// TIA Portal V19 export
FUNCTION_BLOCK "Prod_HMI_Mng"   // FB194, LAD
TITLE = GESTIONE OPERAZIONI ESEGUITE DA HMI
// stored: MemoryReserve 100, SetENOAutomatically false
   VAR_INPUT
      CTRL_LinePreraration : Bool;
      MODE { ExternalAccessible := 'False'; ExternalVisible := 'False'; ExternalWritable := 'False'} : "Prod_Mode";
      PART_PROD { ExternalWritable := 'False'} : "Prod_Part_Area";
      BEAM_PROD { ExternalWritable := 'False'} : "Prod_Beam_Area";
   END_VAR
   VAR_IN_OUT
      SET_UP : "Prod_SetUp_Data";
   END_VAR
   VAR
      i : Int;
      indx_Detail : Int;
      Sts : Struct
         Enable_Pop_ACT_to_TODO : Bool;
         Sel_TODO_CanBeExecuted : Bool;
      END_STRUCT;
      Ctrl : Struct
         Pop_ACT_to_TODO : Bool;
         "Pop_O_ACT_&_Push_O_ENDING" : Bool;
         "Pop_O_TODO_&_Push_O_ACT" : Bool;
         Push_HMI_Order_Push_O_TODO : Bool;
         Move_O_TODO_UP : Bool;
         Move_O_TODO_DW : Bool;
         "Pop_O_TODO_&_Push_O_ENDING" : Bool;
      END_STRUCT;
      TON_HMI_Pop_ACT_To_TODO : TON_TIME;
      TON_HMI_Clear_Index_TODO { S7_SetPoint := 'True'} : TON_TIME;
      TON_HMI_Pop_ACT_To_ENDING { S7_SetPoint := 'True'} : TON_TIME;
      TON_HMI_Pop_TODO_To_ACT { S7_SetPoint := 'True'} : TON_TIME;
      TON_HMI_Pop_TODO_To_ENDING { S7_SetPoint := 'True'} : TON_TIME;
      O_TODO_Push_ManualOrder_HMI { S7_SetPoint := 'True'} : "Prod_O_TODO_Push_ManualOrder";
      O_TODO_Swap_Positions_HMI { S7_SetPoint := 'True'} : "Prod_O_TODO_Swap_Positions";
      SetUp_Man_Mng { S7_SetPoint := 'True'} : "Prod_SetUp_Man";
      AUX : Struct
         Button_Pop_ACT_To_ENDING { ExternalAccessible := 'False'; ExternalVisible := 'False'; ExternalWritable := 'False'} : Bool;
         Button_Pop_ACT_To_TODO { ExternalAccessible := 'False'; ExternalVisible := 'False'; ExternalWritable := 'False'} : Bool;
         Button_Pop_TODO_To_ACT { ExternalAccessible := 'False'; ExternalVisible := 'False'; ExternalWritable := 'False'} : Bool;
         Button_Push_ManualOrder_To_TODO { ExternalAccessible := 'False'; ExternalVisible := 'False'; ExternalWritable := 'False'} : Bool;
         Button_ChangeOrder_TODO_UP { ExternalAccessible := 'False'; ExternalVisible := 'False'; ExternalWritable := 'False'} : Bool;
         Button_ChangeOrder_TODO_DW { ExternalAccessible := 'False'; ExternalVisible := 'False'; ExternalWritable := 'False'} : Bool;
         Button_Pop_TODO_To_ENDING { ExternalAccessible := 'False'; ExternalVisible := 'False'; ExternalWritable := 'False'} : Bool;
         Button_ShowDetatails { ExternalAccessible := 'False'; ExternalVisible := 'False'; ExternalWritable := 'False'} : Bool;
      END_STRUCT;
   END_VAR
   VAR_TEMP
      RETVAL : DInt;
      OK : Bool;
      P_Total : DInt;
      P_Reached_EVEN_Qty : Bool;   // La produzione in corso ha raggiunto un numero pari di SemiGusci
      PE : Struct
         Button_Pop_ACT_To_ENDING : Bool;
         Button_Pop_ACT_To_TODO : Bool;
         Button_Pop_TODO_To_ACT : Bool;
         Button_Push_ManualOrder_To_TODO : Bool;
         Button_ChangeOrder_TODO_UP : Bool;
         Button_ChangeOrder_TODO_DW : Bool;
         Button_Pop_TODO_To_ENDING : Bool;
         Button_ShowDetatails : Bool;
      END_STRUCT;
   END_VAR
   VAR_TEMP   // added for the SCL form of the ladder/FBD networks
      _w1 : Bool;
      _w2 : Bool;
      _w3 : Bool;
      _w4 : Bool;
      _w5 : Bool;
      _w6 : Bool;
      _w7 : Bool;
      _w8 : Bool;
   END_VAR
BEGIN

REGION Network 1 (SCL): <<<HMI >>>

   (*

   # Da HMI si possono fare queste operazioni:

   **Mettere in pausa un ordine in lavoro che era in produzione

   - Se cambio produzione automatico è OFF
   - Se Area (2) è in manuale
   - Se il numero di SemiGusci è pari oppure produzione di pezzi non accoppiati

   **Interrompere un ordine in lavoro spostandolo negli ordini in via di completamente

   - Solo se la macchina è in set up per cancellare eventuali ordini non conclusi

   **Mettere in lavoro un ordine della lista

   - Solo se è impostato che il cambio ordine automatico è OFF
   - Se Area (2) è in manuale
   - Si deve selezionare la riga che si vuole caricare ("Production_HMI".TODO_Index > 1)


   ** Aggiungere un ordine di lavoro che non arriva dal MES (manuale)

   - Se parametro funzionamento MES è messo a OFF
   - Se nella lista non ci sono ordini arrivati dal MES presenti



   ** Cambiare sequenza di esecuzione degli ordini lavoro che non sono arrivati dal MES (manuale)

   - Se parametro funzionamento MES è messo a OFF
   - Se cambio produzione automatico è OFF
   - Se nella lista non ci sono ordini arrivati dal MES presenti

   *)
END_REGION

REGION Network 2: Fronte di salita pulsanti
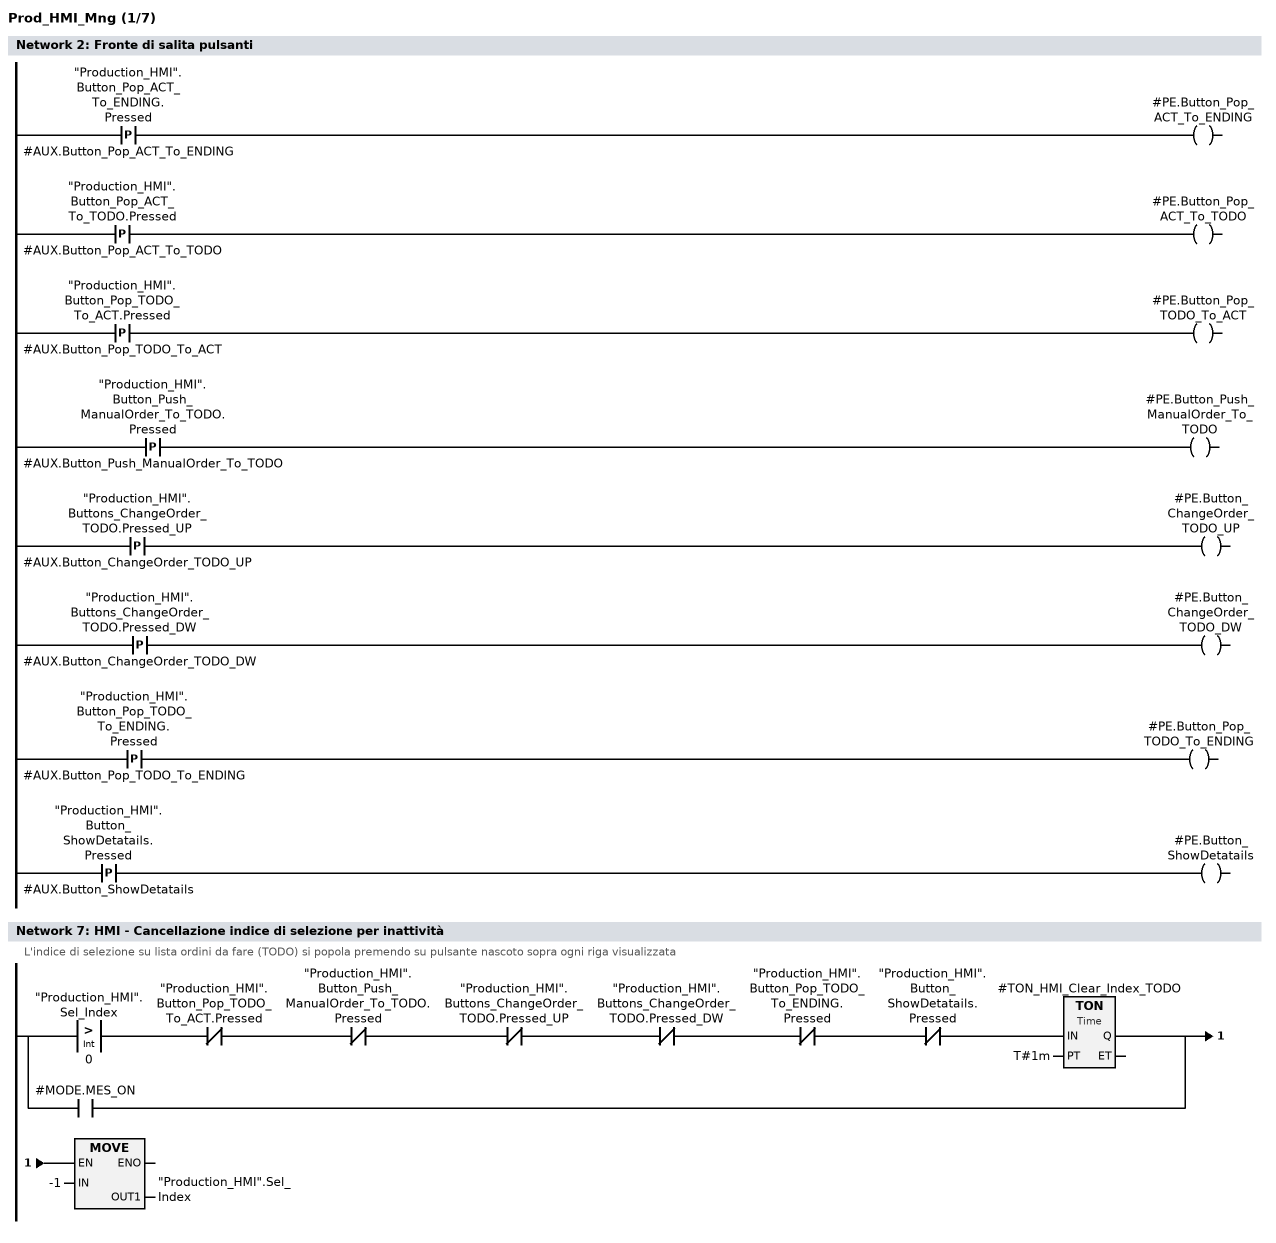
   RUNG wire#powerrail
      P_Contact(operand := "Production_HMI".Button_Pop_ACT_To_ENDING.Pressed, bit := #AUX.Button_Pop_ACT_To_ENDING)
      Coil( #PE.Button_Pop_ACT_To_ENDING )
   END_RUNG
   RUNG wire#powerrail
      P_Contact(operand := "Production_HMI".Button_Pop_ACT_To_TODO.Pressed, bit := #AUX.Button_Pop_ACT_To_TODO)
      Coil( #PE.Button_Pop_ACT_To_TODO )
   END_RUNG
   RUNG wire#powerrail
      P_Contact(operand := "Production_HMI".Button_Pop_TODO_To_ACT.Pressed, bit := #AUX.Button_Pop_TODO_To_ACT)
      Coil( #PE.Button_Pop_TODO_To_ACT )
   END_RUNG
   RUNG wire#powerrail
      P_Contact(operand := "Production_HMI".Button_Push_ManualOrder_To_TODO.Pressed, bit := #AUX.Button_Push_ManualOrder_To_TODO)
      Coil( #PE.Button_Push_ManualOrder_To_TODO )
   END_RUNG
   RUNG wire#powerrail
      P_Contact(operand := "Production_HMI".Buttons_ChangeOrder_TODO.Pressed_UP, bit := #AUX.Button_ChangeOrder_TODO_UP)
      Coil( #PE.Button_ChangeOrder_TODO_UP )
   END_RUNG
   RUNG wire#powerrail
      P_Contact(operand := "Production_HMI".Buttons_ChangeOrder_TODO.Pressed_DW, bit := #AUX.Button_ChangeOrder_TODO_DW)
      Coil( #PE.Button_ChangeOrder_TODO_DW )
   END_RUNG
   RUNG wire#powerrail
      P_Contact(operand := "Production_HMI".Button_Pop_TODO_To_ENDING.Pressed, bit := #AUX.Button_Pop_TODO_To_ENDING)
      Coil( #PE.Button_Pop_TODO_To_ENDING )
   END_RUNG
   RUNG wire#powerrail
      P_Contact(operand := "Production_HMI".Button_ShowDetatails.Pressed, bit := #AUX.Button_ShowDetatails)
      Coil( #PE.Button_ShowDetatails )
   END_RUNG
   // the same network as SCL:
   #_w1 := "Production_HMI".Button_Pop_ACT_To_ENDING.Pressed AND NOT #AUX.Button_Pop_ACT_To_ENDING;   // rising edge of "Production_HMI".Button_Pop_ACT_To_ENDING.Pressed
   #AUX.Button_Pop_ACT_To_ENDING := "Production_HMI".Button_Pop_ACT_To_ENDING.Pressed;
   #PE.Button_Pop_ACT_To_ENDING := #_w1;
   #_w2 := "Production_HMI".Button_Pop_ACT_To_TODO.Pressed AND NOT #AUX.Button_Pop_ACT_To_TODO;   // rising edge of "Production_HMI".Button_Pop_ACT_To_TODO.Pressed
   #AUX.Button_Pop_ACT_To_TODO := "Production_HMI".Button_Pop_ACT_To_TODO.Pressed;
   #PE.Button_Pop_ACT_To_TODO := #_w2;
   #_w3 := "Production_HMI".Button_Pop_TODO_To_ACT.Pressed AND NOT #AUX.Button_Pop_TODO_To_ACT;   // rising edge of "Production_HMI".Button_Pop_TODO_To_ACT.Pressed
   #AUX.Button_Pop_TODO_To_ACT := "Production_HMI".Button_Pop_TODO_To_ACT.Pressed;
   #PE.Button_Pop_TODO_To_ACT := #_w3;
   #_w4 := "Production_HMI".Button_Push_ManualOrder_To_TODO.Pressed AND NOT #AUX.Button_Push_ManualOrder_To_TODO;   // rising edge of "Production_HMI".Button_Push_ManualOrder_To_TODO.Pressed
   #AUX.Button_Push_ManualOrder_To_TODO := "Production_HMI".Button_Push_ManualOrder_To_TODO.Pressed;
   #PE.Button_Push_ManualOrder_To_TODO := #_w4;
   #_w5 := "Production_HMI".Buttons_ChangeOrder_TODO.Pressed_UP AND NOT #AUX.Button_ChangeOrder_TODO_UP;   // rising edge of "Production_HMI".Buttons_ChangeOrder_TODO.Pressed_UP
   #AUX.Button_ChangeOrder_TODO_UP := "Production_HMI".Buttons_ChangeOrder_TODO.Pressed_UP;
   #PE.Button_ChangeOrder_TODO_UP := #_w5;
   #_w6 := "Production_HMI".Buttons_ChangeOrder_TODO.Pressed_DW AND NOT #AUX.Button_ChangeOrder_TODO_DW;   // rising edge of "Production_HMI".Buttons_ChangeOrder_TODO.Pressed_DW
   #AUX.Button_ChangeOrder_TODO_DW := "Production_HMI".Buttons_ChangeOrder_TODO.Pressed_DW;
   #PE.Button_ChangeOrder_TODO_DW := #_w6;
   #_w7 := "Production_HMI".Button_Pop_TODO_To_ENDING.Pressed AND NOT #AUX.Button_Pop_TODO_To_ENDING;   // rising edge of "Production_HMI".Button_Pop_TODO_To_ENDING.Pressed
   #AUX.Button_Pop_TODO_To_ENDING := "Production_HMI".Button_Pop_TODO_To_ENDING.Pressed;
   #PE.Button_Pop_TODO_To_ENDING := #_w7;
   #_w8 := "Production_HMI".Button_ShowDetatails.Pressed AND NOT #AUX.Button_ShowDetatails;   // rising edge of "Production_HMI".Button_ShowDetatails.Pressed
   #AUX.Button_ShowDetatails := "Production_HMI".Button_ShowDetatails.Pressed;
   #PE.Button_ShowDetatails := #_w8;
END_REGION

REGION Network 7: HMI - Cancellazione indice di selezione per inattività
   // L'indice di selezione su lista ordini da fare (TODO) si popola premendo su pulsante nascoto sopra ogni riga visualizzata
   RUNG wire#powerrail
      { S7_Templates := "SrcType := Int" } GT_Contact(in1 := "Production_HMI".Sel_Index, in2 := 0)
      I_Contact( "Production_HMI".Button_Pop_TODO_To_ACT.Pressed )
      I_Contact( "Production_HMI".Button_Push_ManualOrder_To_TODO.Pressed )
      I_Contact( "Production_HMI".Buttons_ChangeOrder_TODO.Pressed_UP )
      I_Contact( "Production_HMI".Buttons_ChangeOrder_TODO.Pressed_DW )
      I_Contact( "Production_HMI".Button_Pop_TODO_To_ENDING.Pressed )
      I_Contact( "Production_HMI".Button_ShowDetatails.Pressed )
      { S7_Templates := "time_type := Time" } #TON_HMI_Clear_Index_TODO.TON(pt := T#1m, et =>)
      wire#w1
      { S7_GenerateENO := "TRUE" } Move(in := -1, out1 => "Production_HMI".Sel_Index)
   END_RUNG
   RUNG wire#powerrail
      Contact( #MODE.MES_ON )
   END_RUNG wire#w1
   // the same network as SCL:
   #TON_HMI_Clear_Index_TODO(IN := ("Production_HMI".Sel_Index > 0) AND NOT "Production_HMI".Button_Pop_TODO_To_ACT.Pressed AND NOT "Production_HMI".Button_Push_ManualOrder_To_TODO.Pressed AND NOT "Production_HMI".Buttons_ChangeOrder_TODO.Pressed_UP AND NOT "Production_HMI".Buttons_ChangeOrder_TODO.Pressed_DW AND NOT "Production_HMI".Button_Pop_TODO_To_ENDING.Pressed AND NOT "Production_HMI".Button_ShowDetatails.Pressed,   // TON
                           PT := T#1m);
   IF #TON_HMI_Clear_Index_TODO.Q OR #MODE.MES_ON THEN "Production_HMI".Sel_Index := -1; END_IF;
END_REGION

REGION Network 8 (SCL): HMI - Ordine in lavoro ha eseguito un numero di parti dispari = Abilitazione a PAUSA ORDINE
   #P_Total := "Production".O_ACT.Parts_GOOD + "Production".O_ACT.Parts_GOOD_R;


   #P_Reached_EVEN_Qty := NOT( (#P_Total MOD 2) <> 0);
END_REGION

REGION Network 9: +
END_REGION

REGION Network 10: < HMI - Ordine (ACT -> TODO) >
END_REGION

REGION Network 11: HMI - Spostamente MANUALE ordine da lavoro a lista ordini da fare (ACT -> TODO) = PAUSA ORDINE INIZIATO
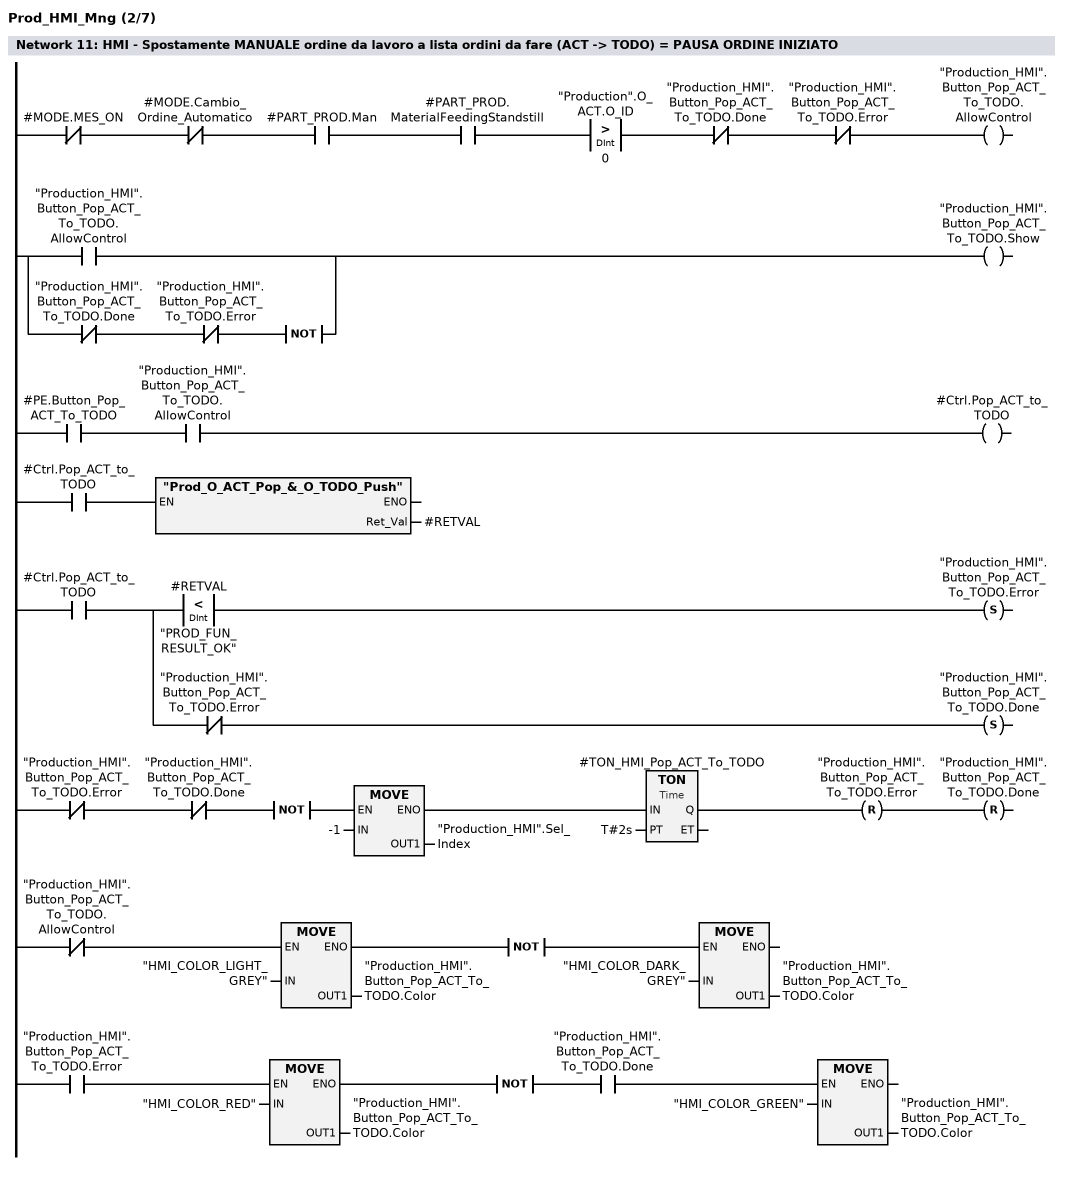
   RUNG wire#powerrail
      I_Contact( #MODE.MES_ON )
      I_Contact( #MODE.Cambio_Ordine_Automatico )
      Contact( #PART_PROD.Man )
      Contact( #PART_PROD.MaterialFeedingStandstill )
      { S7_Templates := "SrcType := DInt" } GT_Contact(in1 := "Production".O_ACT.O_ID, in2 := 0)
      I_Contact( "Production_HMI".Button_Pop_ACT_To_TODO.Done )
      I_Contact( "Production_HMI".Button_Pop_ACT_To_TODO.Error )
      Coil( "Production_HMI".Button_Pop_ACT_To_TODO.AllowControl )
   END_RUNG
   RUNG wire#powerrail
      Contact( "Production_HMI".Button_Pop_ACT_To_TODO.AllowControl )
      wire#w1
      Coil( "Production_HMI".Button_Pop_ACT_To_TODO.Show )
   END_RUNG
   RUNG wire#powerrail
      I_Contact( "Production_HMI".Button_Pop_ACT_To_TODO.Done )
      I_Contact( "Production_HMI".Button_Pop_ACT_To_TODO.Error )
      Not()
   END_RUNG wire#w1
   RUNG wire#powerrail
      Contact( #PE.Button_Pop_ACT_To_TODO )
      Contact( "Production_HMI".Button_Pop_ACT_To_TODO.AllowControl )
      Coil( #Ctrl.Pop_ACT_to_TODO )
   END_RUNG
   RUNG wire#powerrail
      Contact( #Ctrl.Pop_ACT_to_TODO )
      "Prod_O_ACT_Pop_&_O_TODO_Push"(Ret_Val => #RETVAL)
   END_RUNG
   RUNG wire#powerrail
      Contact( #Ctrl.Pop_ACT_to_TODO )
      wire#w2
      { S7_Templates := "SrcType := DInt" } LT_Contact(in1 := #RETVAL, in2 := "PROD_FUN_RESULT_OK")
      S_Coil( "Production_HMI".Button_Pop_ACT_To_TODO.Error )
   END_RUNG
   RUNG wire#w2
      I_Contact( "Production_HMI".Button_Pop_ACT_To_TODO.Error )
      S_Coil( "Production_HMI".Button_Pop_ACT_To_TODO.Done )
   END_RUNG
   RUNG wire#powerrail
      I_Contact( "Production_HMI".Button_Pop_ACT_To_TODO.Error )
      I_Contact( "Production_HMI".Button_Pop_ACT_To_TODO.Done )
      Not()
      { S7_GenerateENO := "TRUE" } Move(in := -1, out1 => "Production_HMI".Sel_Index)
      { S7_Templates := "time_type := Time" } #TON_HMI_Pop_ACT_To_TODO.TON(pt := T#2s, et =>)
      R_Coil( "Production_HMI".Button_Pop_ACT_To_TODO.Error )
      R_Coil( "Production_HMI".Button_Pop_ACT_To_TODO.Done )
   END_RUNG
   RUNG wire#powerrail
      I_Contact( "Production_HMI".Button_Pop_ACT_To_TODO.AllowControl )
      { S7_GenerateENO := "TRUE" } Move(in := "HMI_COLOR_LIGHT_GREY", out1 => "Production_HMI".Button_Pop_ACT_To_TODO.Color)
      Not()
      { S7_GenerateENO := "TRUE" } Move(in := "HMI_COLOR_DARK_GREY", out1 => "Production_HMI".Button_Pop_ACT_To_TODO.Color)
   END_RUNG
   RUNG wire#powerrail
      Contact( "Production_HMI".Button_Pop_ACT_To_TODO.Error )
      { S7_GenerateENO := "TRUE" } Move(in := "HMI_COLOR_RED", out1 => "Production_HMI".Button_Pop_ACT_To_TODO.Color)
      Not()
      Contact( "Production_HMI".Button_Pop_ACT_To_TODO.Done )
      { S7_GenerateENO := "TRUE" } Move(in := "HMI_COLOR_GREEN", out1 => "Production_HMI".Button_Pop_ACT_To_TODO.Color)
   END_RUNG
   // the same network as SCL:
   // ENO of a box is taken as its EN; it also drops when the box reports an error
   "Production_HMI".Button_Pop_ACT_To_TODO.AllowControl := NOT #MODE.MES_ON AND NOT #MODE.Cambio_Ordine_Automatico AND #PART_PROD.Man AND #PART_PROD.MaterialFeedingStandstill AND ("Production".O_ACT.O_ID > 0) AND NOT "Production_HMI".Button_Pop_ACT_To_TODO.Done AND NOT "Production_HMI".Button_Pop_ACT_To_TODO.Error;
   "Production_HMI".Button_Pop_ACT_To_TODO.Show := "Production_HMI".Button_Pop_ACT_To_TODO.AllowControl OR NOT (NOT "Production_HMI".Button_Pop_ACT_To_TODO.Done AND NOT "Production_HMI".Button_Pop_ACT_To_TODO.Error);
   #Ctrl.Pop_ACT_to_TODO := #PE.Button_Pop_ACT_To_TODO AND "Production_HMI".Button_Pop_ACT_To_TODO.AllowControl;
   IF #Ctrl.Pop_ACT_to_TODO THEN #RETVAL := "Prod_O_ACT_Pop_&_O_TODO_Push"(); END_IF;
   IF #Ctrl.Pop_ACT_to_TODO AND (#RETVAL < "PROD_FUN_RESULT_OK") THEN
       "Production_HMI".Button_Pop_ACT_To_TODO.Error := TRUE;
   END_IF;
   IF #Ctrl.Pop_ACT_to_TODO AND NOT "Production_HMI".Button_Pop_ACT_To_TODO.Error THEN
       "Production_HMI".Button_Pop_ACT_To_TODO.Done := TRUE;
   END_IF;
   #_w1 := NOT (NOT "Production_HMI".Button_Pop_ACT_To_TODO.Error AND NOT "Production_HMI".Button_Pop_ACT_To_TODO.Done);
   IF #_w1 THEN "Production_HMI".Sel_Index := -1; END_IF;
   #TON_HMI_Pop_ACT_To_TODO(IN := #_w1, PT := T#2s);   // TON
   IF #TON_HMI_Pop_ACT_To_TODO.Q THEN
       "Production_HMI".Button_Pop_ACT_To_TODO.Error := FALSE;
       "Production_HMI".Button_Pop_ACT_To_TODO.Done := FALSE;
   END_IF;
   #_w2 := NOT "Production_HMI".Button_Pop_ACT_To_TODO.AllowControl;
   IF #_w2 THEN "Production_HMI".Button_Pop_ACT_To_TODO.Color := "HMI_COLOR_LIGHT_GREY"; END_IF;
   IF NOT #_w2 THEN "Production_HMI".Button_Pop_ACT_To_TODO.Color := "HMI_COLOR_DARK_GREY"; END_IF;
   IF "Production_HMI".Button_Pop_ACT_To_TODO.Error THEN
       "Production_HMI".Button_Pop_ACT_To_TODO.Color := "HMI_COLOR_RED";
   END_IF;
   IF NOT "Production_HMI".Button_Pop_ACT_To_TODO.Error AND "Production_HMI".Button_Pop_ACT_To_TODO.Done THEN
       "Production_HMI".Button_Pop_ACT_To_TODO.Color := "HMI_COLOR_GREEN";
   END_IF;
END_REGION

REGION Network 12: +
END_REGION

REGION Network 13: +
END_REGION

REGION Network 14: HMI - Spostamente MANUALE ordine da lavoro a ordini in via di completamento (ACT -> ENDING)
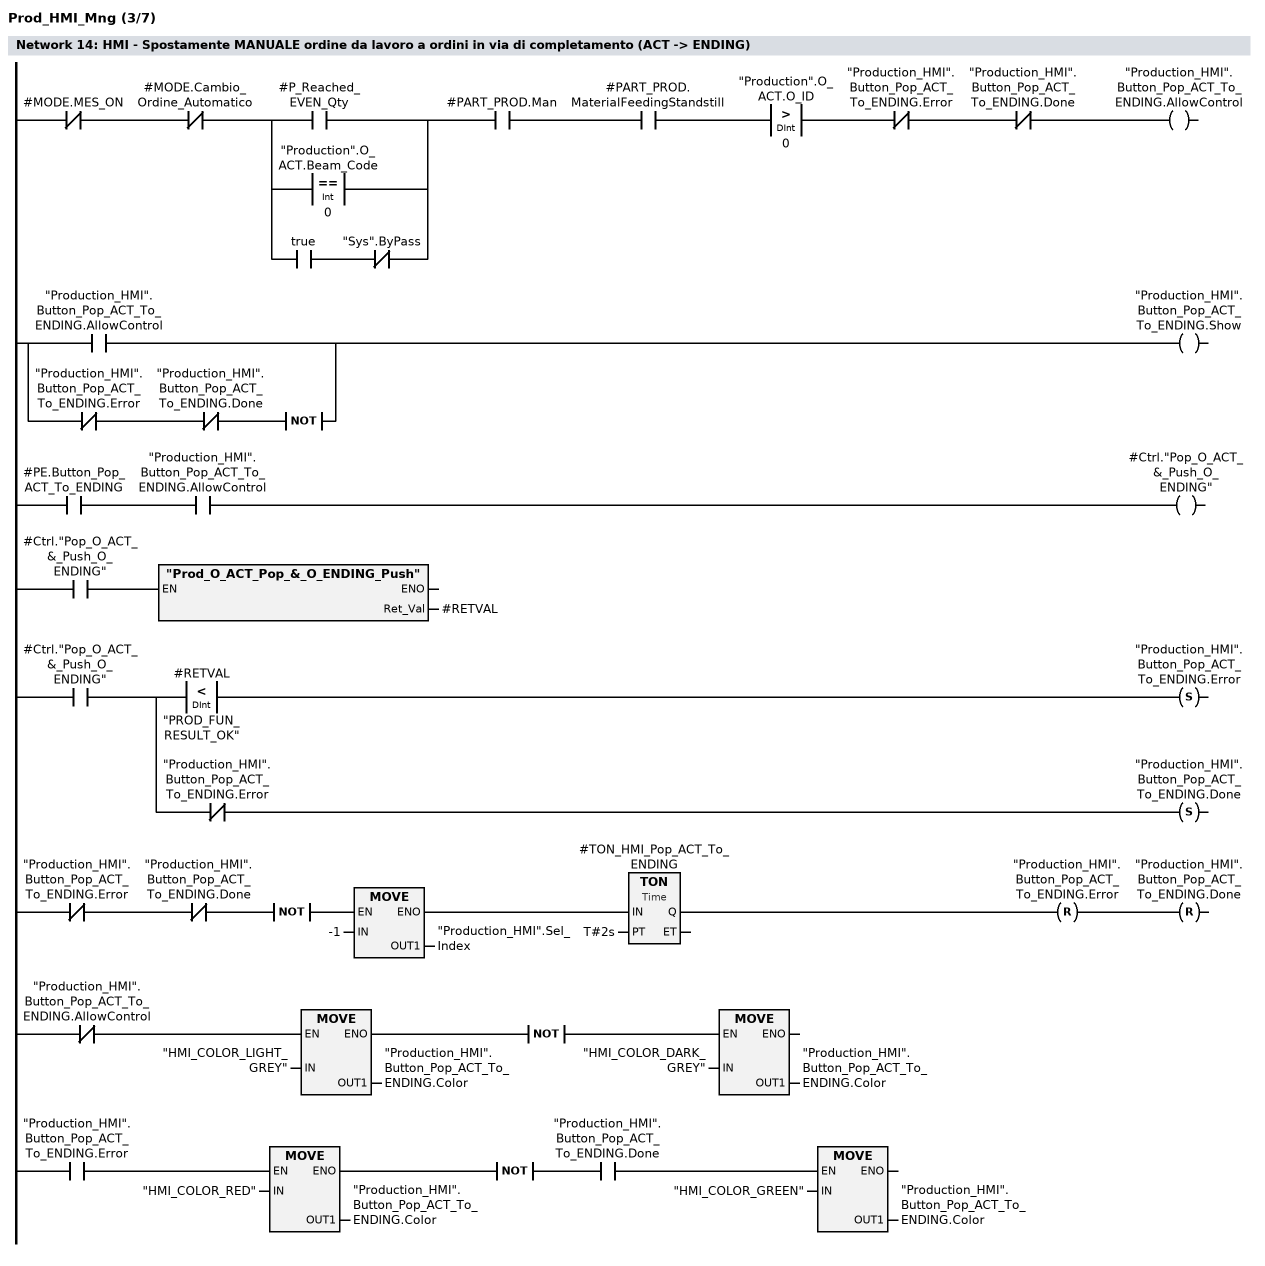
   RUNG wire#powerrail
      I_Contact( #MODE.MES_ON )
      I_Contact( #MODE.Cambio_Ordine_Automatico )
      wire#w1
      Contact( #P_Reached_EVEN_Qty )
      wire#w2
      Contact( #PART_PROD.Man )
      Contact( #PART_PROD.MaterialFeedingStandstill )
      { S7_Templates := "SrcType := DInt" } GT_Contact(in1 := "Production".O_ACT.O_ID, in2 := 0)
      I_Contact( "Production_HMI".Button_Pop_ACT_To_ENDING.Error )
      I_Contact( "Production_HMI".Button_Pop_ACT_To_ENDING.Done )
      Coil( "Production_HMI".Button_Pop_ACT_To_ENDING.AllowControl )
   END_RUNG
   RUNG wire#w1
      { S7_Templates := "SrcType := Int" } EQ_Contact(in1 := "Production".O_ACT.Beam_Code, in2 := 0)
   END_RUNG wire#w2
   RUNG wire#w1
      Contact( true )
      I_Contact( "Sys".ByPass )
   END_RUNG wire#w2
   RUNG wire#powerrail
      Contact( "Production_HMI".Button_Pop_ACT_To_ENDING.AllowControl )
      wire#w3
      Coil( "Production_HMI".Button_Pop_ACT_To_ENDING.Show )
   END_RUNG
   RUNG wire#powerrail
      I_Contact( "Production_HMI".Button_Pop_ACT_To_ENDING.Error )
      I_Contact( "Production_HMI".Button_Pop_ACT_To_ENDING.Done )
      Not()
   END_RUNG wire#w3
   RUNG wire#powerrail
      Contact( #PE.Button_Pop_ACT_To_ENDING )
      Contact( "Production_HMI".Button_Pop_ACT_To_ENDING.AllowControl )
      Coil( #Ctrl."Pop_O_ACT_&_Push_O_ENDING" )
   END_RUNG
   RUNG wire#powerrail
      Contact( #Ctrl."Pop_O_ACT_&_Push_O_ENDING" )
      "Prod_O_ACT_Pop_&_O_ENDING_Push"(Ret_Val => #RETVAL)
   END_RUNG
   RUNG wire#powerrail
      Contact( #Ctrl."Pop_O_ACT_&_Push_O_ENDING" )
      wire#w4
      { S7_Templates := "SrcType := DInt" } LT_Contact(in1 := #RETVAL, in2 := "PROD_FUN_RESULT_OK")
      S_Coil( "Production_HMI".Button_Pop_ACT_To_ENDING.Error )
   END_RUNG
   RUNG wire#w4
      I_Contact( "Production_HMI".Button_Pop_ACT_To_ENDING.Error )
      S_Coil( "Production_HMI".Button_Pop_ACT_To_ENDING.Done )
   END_RUNG
   RUNG wire#powerrail
      I_Contact( "Production_HMI".Button_Pop_ACT_To_ENDING.Error )
      I_Contact( "Production_HMI".Button_Pop_ACT_To_ENDING.Done )
      Not()
      { S7_GenerateENO := "TRUE" } Move(in := -1, out1 => "Production_HMI".Sel_Index)
      { S7_Templates := "time_type := Time" } #TON_HMI_Pop_ACT_To_ENDING.TON(pt := T#2s, et =>)
      R_Coil( "Production_HMI".Button_Pop_ACT_To_ENDING.Error )
      R_Coil( "Production_HMI".Button_Pop_ACT_To_ENDING.Done )
   END_RUNG
   RUNG wire#powerrail
      I_Contact( "Production_HMI".Button_Pop_ACT_To_ENDING.AllowControl )
      { S7_GenerateENO := "TRUE" } Move(in := "HMI_COLOR_LIGHT_GREY", out1 => "Production_HMI".Button_Pop_ACT_To_ENDING.Color)
      Not()
      { S7_GenerateENO := "TRUE" } Move(in := "HMI_COLOR_DARK_GREY", out1 => "Production_HMI".Button_Pop_ACT_To_ENDING.Color)
   END_RUNG
   RUNG wire#powerrail
      Contact( "Production_HMI".Button_Pop_ACT_To_ENDING.Error )
      { S7_GenerateENO := "TRUE" } Move(in := "HMI_COLOR_RED", out1 => "Production_HMI".Button_Pop_ACT_To_ENDING.Color)
      Not()
      Contact( "Production_HMI".Button_Pop_ACT_To_ENDING.Done )
      { S7_GenerateENO := "TRUE" } Move(in := "HMI_COLOR_GREEN", out1 => "Production_HMI".Button_Pop_ACT_To_ENDING.Color)
   END_RUNG
   // the same network as SCL:
   // ENO of a box is taken as its EN; it also drops when the box reports an error
   "Production_HMI".Button_Pop_ACT_To_ENDING.AllowControl := NOT #MODE.MES_ON AND NOT #MODE.Cambio_Ordine_Automatico AND (#P_Reached_EVEN_Qty OR ("Production".O_ACT.Beam_Code = 0) OR (true AND NOT "Sys".ByPass)) AND #PART_PROD.Man AND #PART_PROD.MaterialFeedingStandstill AND ("Production".O_ACT.O_ID > 0) AND NOT "Production_HMI".Button_Pop_ACT_To_ENDING.Error AND NOT "Production_HMI".Button_Pop_ACT_To_ENDING.Done;
   "Production_HMI".Button_Pop_ACT_To_ENDING.Show := "Production_HMI".Button_Pop_ACT_To_ENDING.AllowControl OR NOT (NOT "Production_HMI".Button_Pop_ACT_To_ENDING.Error AND NOT "Production_HMI".Button_Pop_ACT_To_ENDING.Done);
   #Ctrl."Pop_O_ACT_&_Push_O_ENDING" := #PE.Button_Pop_ACT_To_ENDING AND "Production_HMI".Button_Pop_ACT_To_ENDING.AllowControl;
   IF #Ctrl."Pop_O_ACT_&_Push_O_ENDING" THEN #RETVAL := "Prod_O_ACT_Pop_&_O_ENDING_Push"(); END_IF;
   IF #Ctrl."Pop_O_ACT_&_Push_O_ENDING" AND (#RETVAL < "PROD_FUN_RESULT_OK") THEN
       "Production_HMI".Button_Pop_ACT_To_ENDING.Error := TRUE;
   END_IF;
   IF #Ctrl."Pop_O_ACT_&_Push_O_ENDING" AND NOT "Production_HMI".Button_Pop_ACT_To_ENDING.Error THEN
       "Production_HMI".Button_Pop_ACT_To_ENDING.Done := TRUE;
   END_IF;
   #_w1 := NOT (NOT "Production_HMI".Button_Pop_ACT_To_ENDING.Error AND NOT "Production_HMI".Button_Pop_ACT_To_ENDING.Done);
   IF #_w1 THEN "Production_HMI".Sel_Index := -1; END_IF;
   #TON_HMI_Pop_ACT_To_ENDING(IN := #_w1, PT := T#2s);   // TON
   IF #TON_HMI_Pop_ACT_To_ENDING.Q THEN
       "Production_HMI".Button_Pop_ACT_To_ENDING.Error := FALSE;
       "Production_HMI".Button_Pop_ACT_To_ENDING.Done := FALSE;
   END_IF;
   #_w2 := NOT "Production_HMI".Button_Pop_ACT_To_ENDING.AllowControl;
   IF #_w2 THEN "Production_HMI".Button_Pop_ACT_To_ENDING.Color := "HMI_COLOR_LIGHT_GREY"; END_IF;
   IF NOT #_w2 THEN "Production_HMI".Button_Pop_ACT_To_ENDING.Color := "HMI_COLOR_DARK_GREY"; END_IF;
   IF "Production_HMI".Button_Pop_ACT_To_ENDING.Error THEN
       "Production_HMI".Button_Pop_ACT_To_ENDING.Color := "HMI_COLOR_RED";
   END_IF;
   IF NOT "Production_HMI".Button_Pop_ACT_To_ENDING.Error AND "Production_HMI".Button_Pop_ACT_To_ENDING.Done THEN
       "Production_HMI".Button_Pop_ACT_To_ENDING.Color := "HMI_COLOR_GREEN";
   END_IF;
END_REGION

REGION Network 15: +
END_REGION

REGION Network 16: +
END_REGION

REGION Network 17: +
END_REGION

REGION Network 18 (SCL): HMI - Verifica se ordine selezionato è dello stesso PPrf con cui la linea è stata preparata
   #Sts.Sel_TODO_CanBeExecuted := FALSE;


   IF "Production_HMI".Sel_Index >= 1 AND "Production_HMI".Sel_Index <= "PROD_TODO_ITEMS" THEN

       #RETVAL := "Prod_Item_Check_CanGoinProduction"("Production".O_TODO["Production_HMI".Sel_Index]);

       #Sts.Sel_TODO_CanBeExecuted := #RETVAL >= "PROD_FUN_RESULT_OK";

   END_IF;

   #RETVAL := "Prod_Item_Check_CanGoinProduction"("Production".O_TODO[1]);
END_REGION

REGION Network 19: HMI - Spostamente MANUALE ordine da lista ordini da fare a ordine in Lavoro (TODO -> ACT)
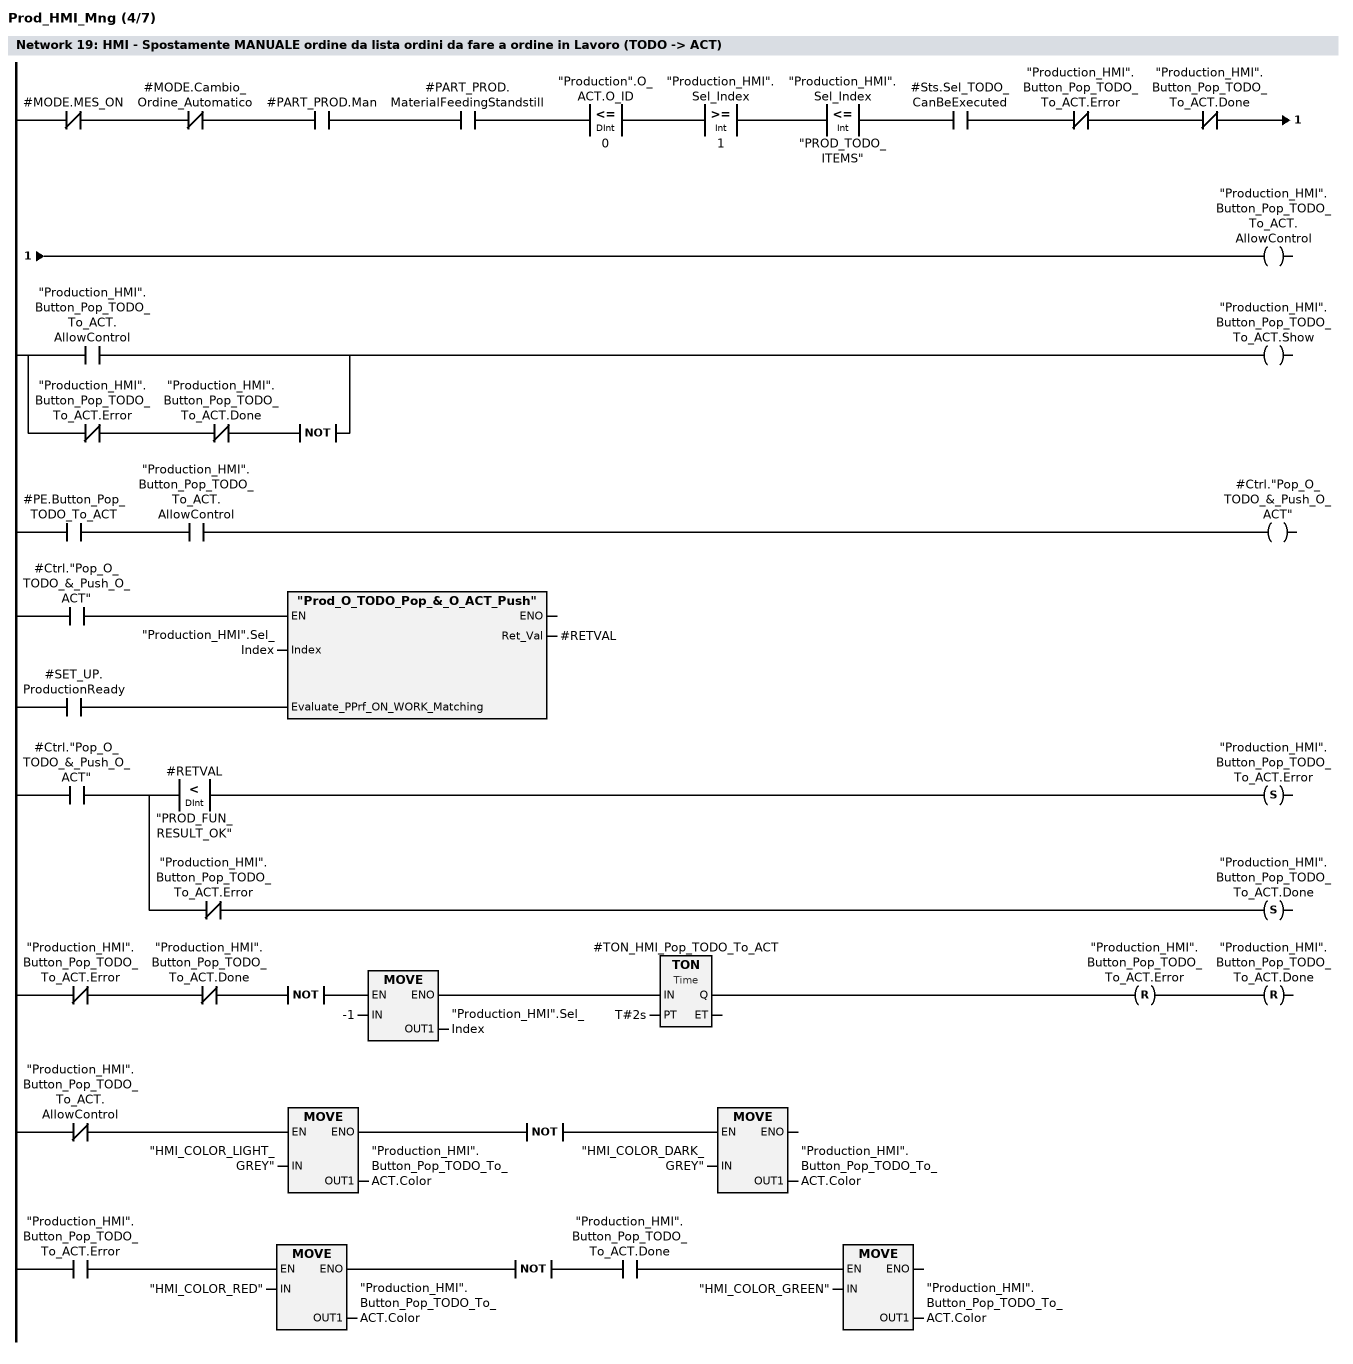
   RUNG wire#powerrail
      I_Contact( #MODE.MES_ON )
      I_Contact( #MODE.Cambio_Ordine_Automatico )
      Contact( #PART_PROD.Man )
      Contact( #PART_PROD.MaterialFeedingStandstill )
      { S7_Templates := "SrcType := DInt" } LE_Contact(in1 := "Production".O_ACT.O_ID, in2 := 0)
      { S7_Templates := "SrcType := Int" } GE_Contact(in1 := "Production_HMI".Sel_Index, in2 := 1)
      { S7_Templates := "SrcType := Int" } LE_Contact(in1 := "Production_HMI".Sel_Index, in2 := "PROD_TODO_ITEMS")
      Contact( #Sts.Sel_TODO_CanBeExecuted )
      I_Contact( "Production_HMI".Button_Pop_TODO_To_ACT.Error )
      I_Contact( "Production_HMI".Button_Pop_TODO_To_ACT.Done )
      Coil( "Production_HMI".Button_Pop_TODO_To_ACT.AllowControl )
   END_RUNG
   RUNG wire#powerrail
      Contact( "Production_HMI".Button_Pop_TODO_To_ACT.AllowControl )
      wire#w1
      Coil( "Production_HMI".Button_Pop_TODO_To_ACT.Show )
   END_RUNG
   RUNG wire#powerrail
      I_Contact( "Production_HMI".Button_Pop_TODO_To_ACT.Error )
      I_Contact( "Production_HMI".Button_Pop_TODO_To_ACT.Done )
      Not()
   END_RUNG wire#w1
   RUNG wire#powerrail
      Contact( #PE.Button_Pop_TODO_To_ACT )
      Contact( "Production_HMI".Button_Pop_TODO_To_ACT.AllowControl )
      Coil( #Ctrl."Pop_O_TODO_&_Push_O_ACT" )
   END_RUNG
   RUNG wire#powerrail
      Contact( #Ctrl."Pop_O_TODO_&_Push_O_ACT" )
      "Prod_O_TODO_Pop_&_O_ACT_Push"(Evaluate_PPrf_ON_WORK_Matching := wire#w2, Index := "Production_HMI".Sel_Index, Ret_Val => #RETVAL)
   END_RUNG
   RUNG wire#powerrail
      Contact( #SET_UP.ProductionReady )
   END_RUNG wire#w2
   RUNG wire#powerrail
      Contact( #Ctrl."Pop_O_TODO_&_Push_O_ACT" )
      wire#w3
      { S7_Templates := "SrcType := DInt" } LT_Contact(in1 := #RETVAL, in2 := "PROD_FUN_RESULT_OK")
      S_Coil( "Production_HMI".Button_Pop_TODO_To_ACT.Error )
   END_RUNG
   RUNG wire#w3
      I_Contact( "Production_HMI".Button_Pop_TODO_To_ACT.Error )
      S_Coil( "Production_HMI".Button_Pop_TODO_To_ACT.Done )
   END_RUNG
   RUNG wire#powerrail
      I_Contact( "Production_HMI".Button_Pop_TODO_To_ACT.Error )
      I_Contact( "Production_HMI".Button_Pop_TODO_To_ACT.Done )
      Not()
      { S7_GenerateENO := "TRUE" } Move(in := -1, out1 => "Production_HMI".Sel_Index)
      { S7_Templates := "time_type := Time" } #TON_HMI_Pop_TODO_To_ACT.TON(pt := T#2s, et =>)
      R_Coil( "Production_HMI".Button_Pop_TODO_To_ACT.Error )
      R_Coil( "Production_HMI".Button_Pop_TODO_To_ACT.Done )
   END_RUNG
   RUNG wire#powerrail
      I_Contact( "Production_HMI".Button_Pop_TODO_To_ACT.AllowControl )
      { S7_GenerateENO := "TRUE" } Move(in := "HMI_COLOR_LIGHT_GREY", out1 => "Production_HMI".Button_Pop_TODO_To_ACT.Color)
      Not()
      { S7_GenerateENO := "TRUE" } Move(in := "HMI_COLOR_DARK_GREY", out1 => "Production_HMI".Button_Pop_TODO_To_ACT.Color)
   END_RUNG
   RUNG wire#powerrail
      Contact( "Production_HMI".Button_Pop_TODO_To_ACT.Error )
      { S7_GenerateENO := "TRUE" } Move(in := "HMI_COLOR_RED", out1 => "Production_HMI".Button_Pop_TODO_To_ACT.Color)
      Not()
      Contact( "Production_HMI".Button_Pop_TODO_To_ACT.Done )
      { S7_GenerateENO := "TRUE" } Move(in := "HMI_COLOR_GREEN", out1 => "Production_HMI".Button_Pop_TODO_To_ACT.Color)
   END_RUNG
   // the same network as SCL:
   // ENO of a box is taken as its EN; it also drops when the box reports an error
   "Production_HMI".Button_Pop_TODO_To_ACT.AllowControl := NOT #MODE.MES_ON AND NOT #MODE.Cambio_Ordine_Automatico AND #PART_PROD.Man AND #PART_PROD.MaterialFeedingStandstill AND ("Production".O_ACT.O_ID <= 0) AND ("Production_HMI".Sel_Index >= 1) AND ("Production_HMI".Sel_Index <= "PROD_TODO_ITEMS") AND #Sts.Sel_TODO_CanBeExecuted AND NOT "Production_HMI".Button_Pop_TODO_To_ACT.Error AND NOT "Production_HMI".Button_Pop_TODO_To_ACT.Done;
   "Production_HMI".Button_Pop_TODO_To_ACT.Show := "Production_HMI".Button_Pop_TODO_To_ACT.AllowControl OR NOT (NOT "Production_HMI".Button_Pop_TODO_To_ACT.Error AND NOT "Production_HMI".Button_Pop_TODO_To_ACT.Done);
   #Ctrl."Pop_O_TODO_&_Push_O_ACT" := #PE.Button_Pop_TODO_To_ACT AND "Production_HMI".Button_Pop_TODO_To_ACT.AllowControl;
   IF #Ctrl."Pop_O_TODO_&_Push_O_ACT" THEN
       #RETVAL := "Prod_O_TODO_Pop_&_O_ACT_Push"(Index := "Production_HMI".Sel_Index,
                               Evaluate_PPrf_ON_WORK_Matching := #SET_UP.ProductionReady);
   END_IF;
   IF #Ctrl."Pop_O_TODO_&_Push_O_ACT" AND (#RETVAL < "PROD_FUN_RESULT_OK") THEN
       "Production_HMI".Button_Pop_TODO_To_ACT.Error := TRUE;
   END_IF;
   IF #Ctrl."Pop_O_TODO_&_Push_O_ACT" AND NOT "Production_HMI".Button_Pop_TODO_To_ACT.Error THEN
       "Production_HMI".Button_Pop_TODO_To_ACT.Done := TRUE;
   END_IF;
   #_w1 := NOT (NOT "Production_HMI".Button_Pop_TODO_To_ACT.Error AND NOT "Production_HMI".Button_Pop_TODO_To_ACT.Done);
   IF #_w1 THEN "Production_HMI".Sel_Index := -1; END_IF;
   #TON_HMI_Pop_TODO_To_ACT(IN := #_w1, PT := T#2s);   // TON
   IF #TON_HMI_Pop_TODO_To_ACT.Q THEN
       "Production_HMI".Button_Pop_TODO_To_ACT.Error := FALSE;
       "Production_HMI".Button_Pop_TODO_To_ACT.Done := FALSE;
   END_IF;
   #_w2 := NOT "Production_HMI".Button_Pop_TODO_To_ACT.AllowControl;
   IF #_w2 THEN "Production_HMI".Button_Pop_TODO_To_ACT.Color := "HMI_COLOR_LIGHT_GREY"; END_IF;
   IF NOT #_w2 THEN "Production_HMI".Button_Pop_TODO_To_ACT.Color := "HMI_COLOR_DARK_GREY"; END_IF;
   IF "Production_HMI".Button_Pop_TODO_To_ACT.Error THEN
       "Production_HMI".Button_Pop_TODO_To_ACT.Color := "HMI_COLOR_RED";
   END_IF;
   IF NOT "Production_HMI".Button_Pop_TODO_To_ACT.Error AND "Production_HMI".Button_Pop_TODO_To_ACT.Done THEN
       "Production_HMI".Button_Pop_TODO_To_ACT.Color := "HMI_COLOR_GREEN";
   END_IF;
END_REGION

REGION Network 20: +
END_REGION

REGION Network 21: +
END_REGION

REGION Network 22: +
END_REGION

REGION Network 23: +
END_REGION

REGION Network 24: HMI - Caricamento MANUALE ordine di lavoro su TODO
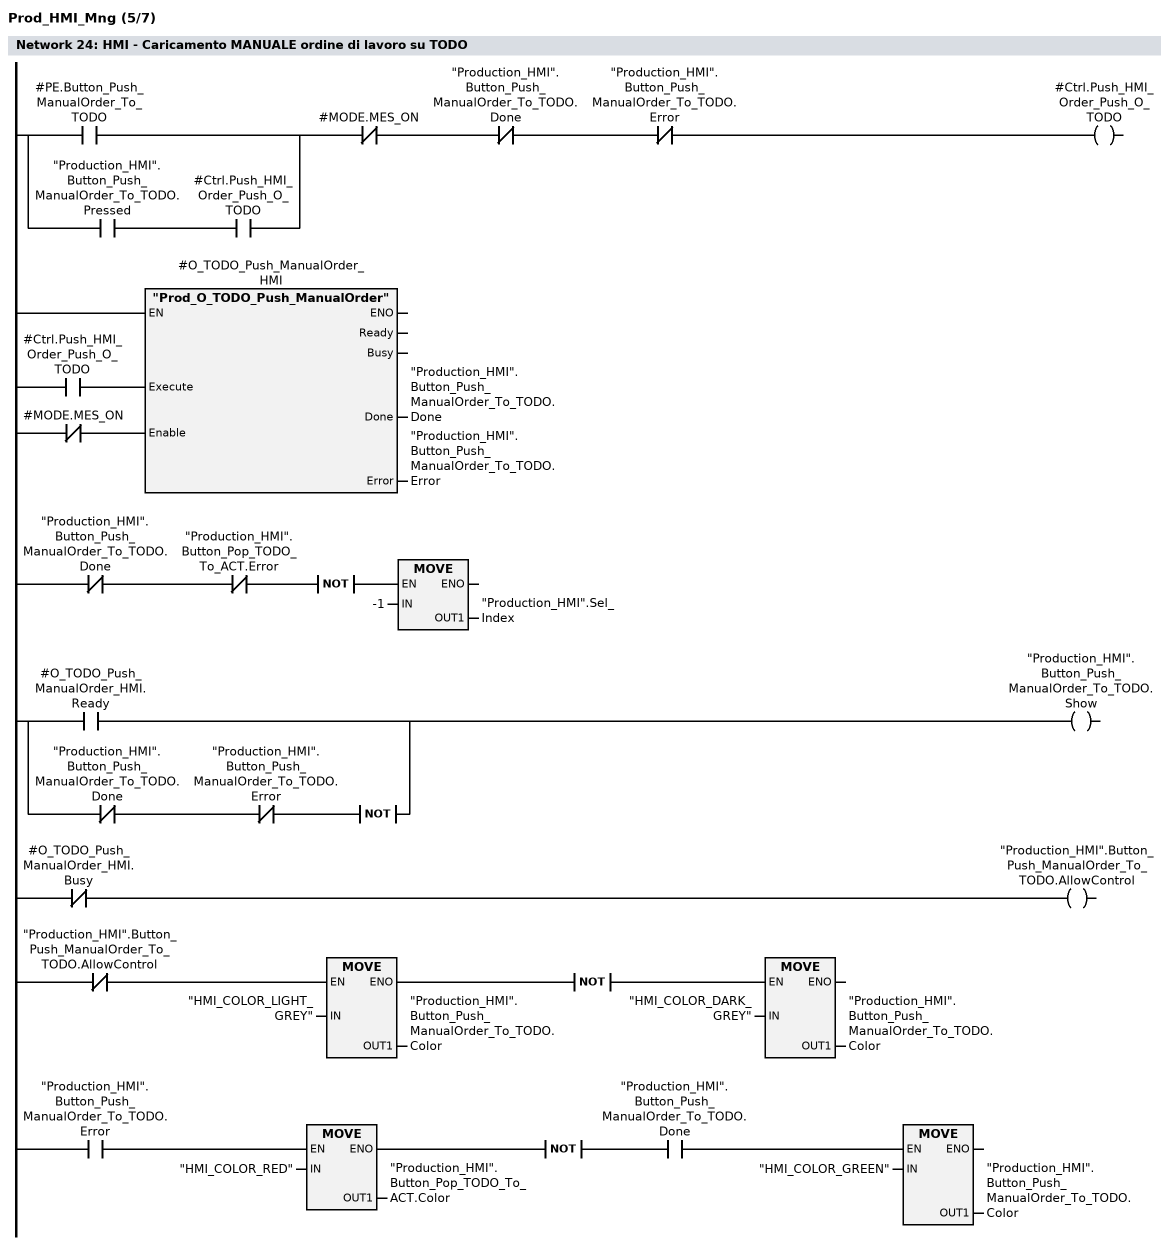
   RUNG wire#powerrail
      Contact( #PE.Button_Push_ManualOrder_To_TODO )
      wire#w1
      I_Contact( #MODE.MES_ON )
      I_Contact( "Production_HMI".Button_Push_ManualOrder_To_TODO.Done )
      I_Contact( "Production_HMI".Button_Push_ManualOrder_To_TODO.Error )
      Coil( #Ctrl.Push_HMI_Order_Push_O_TODO )
   END_RUNG
   RUNG wire#powerrail
      Contact( "Production_HMI".Button_Push_ManualOrder_To_TODO.Pressed )
      Contact( #Ctrl.Push_HMI_Order_Push_O_TODO )
   END_RUNG wire#w1
   RUNG wire#powerrail
      #O_TODO_Push_ManualOrder_HMI(Execute := wire#w2, Enable := wire#w3, Ready =>, Busy =>, Done => "Production_HMI".Button_Push_ManualOrder_To_TODO.Done, Error => "Production_HMI".Button_Push_ManualOrder_To_TODO.Error)
   END_RUNG
   RUNG wire#powerrail
      Contact( #Ctrl.Push_HMI_Order_Push_O_TODO )
   END_RUNG wire#w2
   RUNG wire#powerrail
      I_Contact( #MODE.MES_ON )
   END_RUNG wire#w3
   RUNG wire#powerrail
      I_Contact( "Production_HMI".Button_Push_ManualOrder_To_TODO.Done )
      I_Contact( "Production_HMI".Button_Pop_TODO_To_ACT.Error )
      Not()
      { S7_GenerateENO := "TRUE" } Move(in := -1, out1 => "Production_HMI".Sel_Index)
   END_RUNG
   RUNG wire#powerrail
      Contact( #O_TODO_Push_ManualOrder_HMI.Ready )
      wire#w4
      Coil( "Production_HMI".Button_Push_ManualOrder_To_TODO.Show )
   END_RUNG
   RUNG wire#powerrail
      I_Contact( "Production_HMI".Button_Push_ManualOrder_To_TODO.Done )
      I_Contact( "Production_HMI".Button_Push_ManualOrder_To_TODO.Error )
      Not()
   END_RUNG wire#w4
   RUNG wire#powerrail
      I_Contact( #O_TODO_Push_ManualOrder_HMI.Busy )
      Coil( "Production_HMI".Button_Push_ManualOrder_To_TODO.AllowControl )
   END_RUNG
   RUNG wire#powerrail
      I_Contact( "Production_HMI".Button_Push_ManualOrder_To_TODO.AllowControl )
      { S7_GenerateENO := "TRUE" } Move(in := "HMI_COLOR_LIGHT_GREY", out1 => "Production_HMI".Button_Push_ManualOrder_To_TODO.Color)
      Not()
      { S7_GenerateENO := "TRUE" } Move(in := "HMI_COLOR_DARK_GREY", out1 => "Production_HMI".Button_Push_ManualOrder_To_TODO.Color)
   END_RUNG
   RUNG wire#powerrail
      Contact( "Production_HMI".Button_Push_ManualOrder_To_TODO.Error )
      { S7_GenerateENO := "TRUE" } Move(in := "HMI_COLOR_RED", out1 => "Production_HMI".Button_Pop_TODO_To_ACT.Color)
      Not()
      Contact( "Production_HMI".Button_Push_ManualOrder_To_TODO.Done )
      { S7_GenerateENO := "TRUE" } Move(in := "HMI_COLOR_GREEN", out1 => "Production_HMI".Button_Push_ManualOrder_To_TODO.Color)
   END_RUNG
   // the same network as SCL:
   // ENO of a box is taken as its EN; it also drops when the box reports an error
   #Ctrl.Push_HMI_Order_Push_O_TODO := (#PE.Button_Push_ManualOrder_To_TODO OR ("Production_HMI".Button_Push_ManualOrder_To_TODO.Pressed AND #Ctrl.Push_HMI_Order_Push_O_TODO)) AND NOT #MODE.MES_ON AND NOT "Production_HMI".Button_Push_ManualOrder_To_TODO.Done AND NOT "Production_HMI".Button_Push_ManualOrder_To_TODO.Error;
   #O_TODO_Push_ManualOrder_HMI(Execute := #Ctrl.Push_HMI_Order_Push_O_TODO,   // "Prod_O_TODO_Push_ManualOrder"
                           Enable := NOT #MODE.MES_ON,
                           Done => "Production_HMI".Button_Push_ManualOrder_To_TODO.Done,
                           Error => "Production_HMI".Button_Push_ManualOrder_To_TODO.Error);
   IF NOT (NOT "Production_HMI".Button_Push_ManualOrder_To_TODO.Done AND NOT "Production_HMI".Button_Pop_TODO_To_ACT.Error) THEN
       "Production_HMI".Sel_Index := -1;
   END_IF;
   "Production_HMI".Button_Push_ManualOrder_To_TODO.Show := #O_TODO_Push_ManualOrder_HMI.Ready OR NOT (NOT "Production_HMI".Button_Push_ManualOrder_To_TODO.Done AND NOT "Production_HMI".Button_Push_ManualOrder_To_TODO.Error);
   "Production_HMI".Button_Push_ManualOrder_To_TODO.AllowControl := NOT #O_TODO_Push_ManualOrder_HMI.Busy;
   #_w1 := NOT "Production_HMI".Button_Push_ManualOrder_To_TODO.AllowControl;
   IF #_w1 THEN "Production_HMI".Button_Push_ManualOrder_To_TODO.Color := "HMI_COLOR_LIGHT_GREY"; END_IF;
   IF NOT #_w1 THEN "Production_HMI".Button_Push_ManualOrder_To_TODO.Color := "HMI_COLOR_DARK_GREY"; END_IF;
   IF "Production_HMI".Button_Push_ManualOrder_To_TODO.Error THEN
       "Production_HMI".Button_Pop_TODO_To_ACT.Color := "HMI_COLOR_RED";
   END_IF;
   IF NOT "Production_HMI".Button_Push_ManualOrder_To_TODO.Error AND "Production_HMI".Button_Push_ManualOrder_To_TODO.Done THEN
       "Production_HMI".Button_Push_ManualOrder_To_TODO.Color := "HMI_COLOR_GREEN";
   END_IF;
END_REGION

REGION Network 25: HMI - Cambio ordine di esecuzione degli ordini su TODO
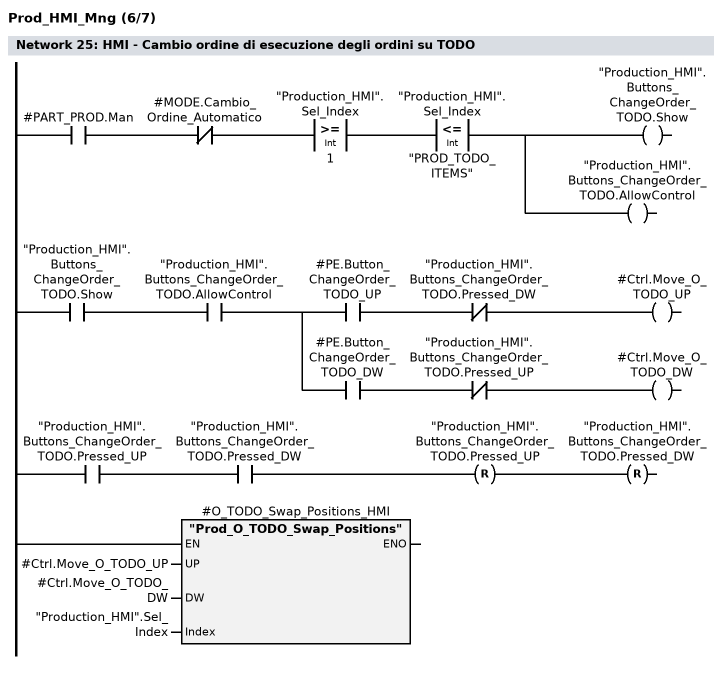
   RUNG wire#powerrail
      Contact( #PART_PROD.Man )
      I_Contact( #MODE.Cambio_Ordine_Automatico )
      { S7_Templates := "SrcType := Int" } GE_Contact(in1 := "Production_HMI".Sel_Index, in2 := 1)
      { S7_Templates := "SrcType := Int" } LE_Contact(in1 := "Production_HMI".Sel_Index, in2 := "PROD_TODO_ITEMS")
      wire#w1
      Coil( "Production_HMI".Buttons_ChangeOrder_TODO.Show )
   END_RUNG
   RUNG wire#w1
      Coil( "Production_HMI".Buttons_ChangeOrder_TODO.AllowControl )
   END_RUNG
   RUNG wire#powerrail
      Contact( "Production_HMI".Buttons_ChangeOrder_TODO.Show )
      Contact( "Production_HMI".Buttons_ChangeOrder_TODO.AllowControl )
      wire#w2
      Contact( #PE.Button_ChangeOrder_TODO_UP )
      I_Contact( "Production_HMI".Buttons_ChangeOrder_TODO.Pressed_DW )
      Coil( #Ctrl.Move_O_TODO_UP )
   END_RUNG
   RUNG wire#w2
      Contact( #PE.Button_ChangeOrder_TODO_DW )
      I_Contact( "Production_HMI".Buttons_ChangeOrder_TODO.Pressed_UP )
      Coil( #Ctrl.Move_O_TODO_DW )
   END_RUNG
   RUNG wire#powerrail
      Contact( "Production_HMI".Buttons_ChangeOrder_TODO.Pressed_UP )
      Contact( "Production_HMI".Buttons_ChangeOrder_TODO.Pressed_DW )
      R_Coil( "Production_HMI".Buttons_ChangeOrder_TODO.Pressed_UP )
      R_Coil( "Production_HMI".Buttons_ChangeOrder_TODO.Pressed_DW )
   END_RUNG
   RUNG wire#powerrail
      #O_TODO_Swap_Positions_HMI(UP := #Ctrl.Move_O_TODO_UP, DW := #Ctrl.Move_O_TODO_DW, Index := "Production_HMI".Sel_Index)
   END_RUNG
   // the same network as SCL:
   "Production_HMI".Buttons_ChangeOrder_TODO.Show := #PART_PROD.Man AND NOT #MODE.Cambio_Ordine_Automatico AND ("Production_HMI".Sel_Index >= 1) AND ("Production_HMI".Sel_Index <= "PROD_TODO_ITEMS");
   "Production_HMI".Buttons_ChangeOrder_TODO.AllowControl := "Production_HMI".Buttons_ChangeOrder_TODO.Show;
   #_w1 := "Production_HMI".Buttons_ChangeOrder_TODO.Show AND "Production_HMI".Buttons_ChangeOrder_TODO.AllowControl;
   #Ctrl.Move_O_TODO_UP := #_w1 AND #PE.Button_ChangeOrder_TODO_UP AND NOT "Production_HMI".Buttons_ChangeOrder_TODO.Pressed_DW;
   #Ctrl.Move_O_TODO_DW := #_w1 AND #PE.Button_ChangeOrder_TODO_DW AND NOT "Production_HMI".Buttons_ChangeOrder_TODO.Pressed_UP;
   #_w2 := "Production_HMI".Buttons_ChangeOrder_TODO.Pressed_UP AND "Production_HMI".Buttons_ChangeOrder_TODO.Pressed_DW;
   IF #_w2 THEN
       "Production_HMI".Buttons_ChangeOrder_TODO.Pressed_UP := FALSE;
       "Production_HMI".Buttons_ChangeOrder_TODO.Pressed_DW := FALSE;
   END_IF;
   #O_TODO_Swap_Positions_HMI(UP := #Ctrl.Move_O_TODO_UP,   // "Prod_O_TODO_Swap_Positions"
                           DW := #Ctrl.Move_O_TODO_DW,
                           Index := "Production_HMI".Sel_Index);
END_REGION

REGION Network 26: HMI - Pop ordine da lista ordine da fare a ordini in via di completamento (TODO -> ENDING)
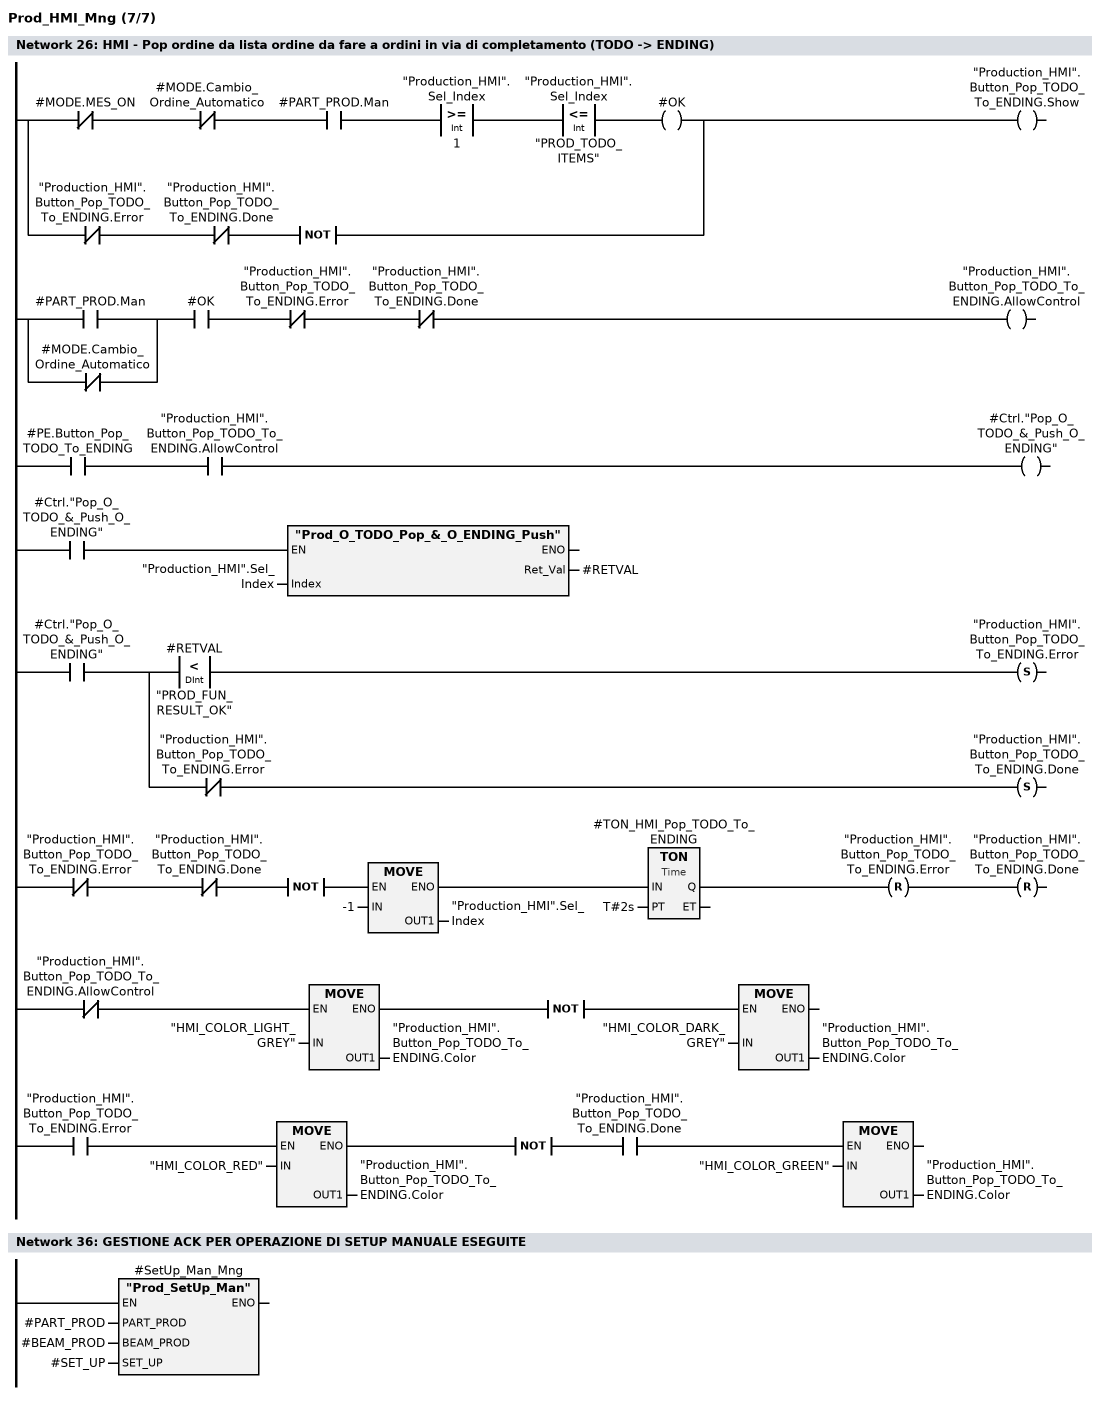
   RUNG wire#powerrail
      I_Contact( #MODE.MES_ON )
      I_Contact( #MODE.Cambio_Ordine_Automatico )
      Contact( #PART_PROD.Man )
      { S7_Templates := "SrcType := Int" } GE_Contact(in1 := "Production_HMI".Sel_Index, in2 := 1)
      { S7_Templates := "SrcType := Int" } LE_Contact(in1 := "Production_HMI".Sel_Index, in2 := "PROD_TODO_ITEMS")
      Coil( #OK )
      wire#w1
      Coil( "Production_HMI".Button_Pop_TODO_To_ENDING.Show )
   END_RUNG
   RUNG wire#powerrail
      I_Contact( "Production_HMI".Button_Pop_TODO_To_ENDING.Error )
      I_Contact( "Production_HMI".Button_Pop_TODO_To_ENDING.Done )
      Not()
   END_RUNG wire#w1
   RUNG wire#powerrail
      Contact( #PART_PROD.Man )
      wire#w2
      Contact( #OK )
      I_Contact( "Production_HMI".Button_Pop_TODO_To_ENDING.Error )
      I_Contact( "Production_HMI".Button_Pop_TODO_To_ENDING.Done )
      Coil( "Production_HMI".Button_Pop_TODO_To_ENDING.AllowControl )
   END_RUNG
   RUNG wire#powerrail
      I_Contact( #MODE.Cambio_Ordine_Automatico )
   END_RUNG wire#w2
   RUNG wire#powerrail
      Contact( #PE.Button_Pop_TODO_To_ENDING )
      Contact( "Production_HMI".Button_Pop_TODO_To_ENDING.AllowControl )
      Coil( #Ctrl."Pop_O_TODO_&_Push_O_ENDING" )
   END_RUNG
   RUNG wire#powerrail
      Contact( #Ctrl."Pop_O_TODO_&_Push_O_ENDING" )
      "Prod_O_TODO_Pop_&_O_ENDING_Push"(Index := "Production_HMI".Sel_Index, Ret_Val => #RETVAL)
   END_RUNG
   RUNG wire#powerrail
      Contact( #Ctrl."Pop_O_TODO_&_Push_O_ENDING" )
      wire#w3
      { S7_Templates := "SrcType := DInt" } LT_Contact(in1 := #RETVAL, in2 := "PROD_FUN_RESULT_OK")
      S_Coil( "Production_HMI".Button_Pop_TODO_To_ENDING.Error )
   END_RUNG
   RUNG wire#w3
      I_Contact( "Production_HMI".Button_Pop_TODO_To_ENDING.Error )
      S_Coil( "Production_HMI".Button_Pop_TODO_To_ENDING.Done )
   END_RUNG
   RUNG wire#powerrail
      I_Contact( "Production_HMI".Button_Pop_TODO_To_ENDING.Error )
      I_Contact( "Production_HMI".Button_Pop_TODO_To_ENDING.Done )
      Not()
      { S7_GenerateENO := "TRUE" } Move(in := -1, out1 => "Production_HMI".Sel_Index)
      { S7_Templates := "time_type := Time" } #TON_HMI_Pop_TODO_To_ENDING.TON(pt := T#2s, et =>)
      R_Coil( "Production_HMI".Button_Pop_TODO_To_ENDING.Error )
      R_Coil( "Production_HMI".Button_Pop_TODO_To_ENDING.Done )
   END_RUNG
   RUNG wire#powerrail
      I_Contact( "Production_HMI".Button_Pop_TODO_To_ENDING.AllowControl )
      { S7_GenerateENO := "TRUE" } Move(in := "HMI_COLOR_LIGHT_GREY", out1 => "Production_HMI".Button_Pop_TODO_To_ENDING.Color)
      Not()
      { S7_GenerateENO := "TRUE" } Move(in := "HMI_COLOR_DARK_GREY", out1 => "Production_HMI".Button_Pop_TODO_To_ENDING.Color)
   END_RUNG
   RUNG wire#powerrail
      Contact( "Production_HMI".Button_Pop_TODO_To_ENDING.Error )
      { S7_GenerateENO := "TRUE" } Move(in := "HMI_COLOR_RED", out1 => "Production_HMI".Button_Pop_TODO_To_ENDING.Color)
      Not()
      Contact( "Production_HMI".Button_Pop_TODO_To_ENDING.Done )
      { S7_GenerateENO := "TRUE" } Move(in := "HMI_COLOR_GREEN", out1 => "Production_HMI".Button_Pop_TODO_To_ENDING.Color)
   END_RUNG
   // the same network as SCL:
   // ENO of a box is taken as its EN; it also drops when the box reports an error
   #OK := NOT #MODE.MES_ON AND NOT #MODE.Cambio_Ordine_Automatico AND #PART_PROD.Man AND ("Production_HMI".Sel_Index >= 1) AND ("Production_HMI".Sel_Index <= "PROD_TODO_ITEMS");
   "Production_HMI".Button_Pop_TODO_To_ENDING.Show := #OK OR NOT (NOT "Production_HMI".Button_Pop_TODO_To_ENDING.Error AND NOT "Production_HMI".Button_Pop_TODO_To_ENDING.Done);
   "Production_HMI".Button_Pop_TODO_To_ENDING.AllowControl := (#PART_PROD.Man OR NOT #MODE.Cambio_Ordine_Automatico) AND #OK AND NOT "Production_HMI".Button_Pop_TODO_To_ENDING.Error AND NOT "Production_HMI".Button_Pop_TODO_To_ENDING.Done;
   #Ctrl."Pop_O_TODO_&_Push_O_ENDING" := #PE.Button_Pop_TODO_To_ENDING AND "Production_HMI".Button_Pop_TODO_To_ENDING.AllowControl;
   IF #Ctrl."Pop_O_TODO_&_Push_O_ENDING" THEN
       #RETVAL := "Prod_O_TODO_Pop_&_O_ENDING_Push"(Index := "Production_HMI".Sel_Index);
   END_IF;
   IF #Ctrl."Pop_O_TODO_&_Push_O_ENDING" AND (#RETVAL < "PROD_FUN_RESULT_OK") THEN
       "Production_HMI".Button_Pop_TODO_To_ENDING.Error := TRUE;
   END_IF;
   IF #Ctrl."Pop_O_TODO_&_Push_O_ENDING" AND NOT "Production_HMI".Button_Pop_TODO_To_ENDING.Error THEN
       "Production_HMI".Button_Pop_TODO_To_ENDING.Done := TRUE;
   END_IF;
   #_w1 := NOT (NOT "Production_HMI".Button_Pop_TODO_To_ENDING.Error AND NOT "Production_HMI".Button_Pop_TODO_To_ENDING.Done);
   IF #_w1 THEN "Production_HMI".Sel_Index := -1; END_IF;
   #TON_HMI_Pop_TODO_To_ENDING(IN := #_w1, PT := T#2s);   // TON
   IF #TON_HMI_Pop_TODO_To_ENDING.Q THEN
       "Production_HMI".Button_Pop_TODO_To_ENDING.Error := FALSE;
       "Production_HMI".Button_Pop_TODO_To_ENDING.Done := FALSE;
   END_IF;
   #_w2 := NOT "Production_HMI".Button_Pop_TODO_To_ENDING.AllowControl;
   IF #_w2 THEN "Production_HMI".Button_Pop_TODO_To_ENDING.Color := "HMI_COLOR_LIGHT_GREY"; END_IF;
   IF NOT #_w2 THEN "Production_HMI".Button_Pop_TODO_To_ENDING.Color := "HMI_COLOR_DARK_GREY"; END_IF;
   IF "Production_HMI".Button_Pop_TODO_To_ENDING.Error THEN
       "Production_HMI".Button_Pop_TODO_To_ENDING.Color := "HMI_COLOR_RED";
   END_IF;
   IF NOT "Production_HMI".Button_Pop_TODO_To_ENDING.Error AND "Production_HMI".Button_Pop_TODO_To_ENDING.Done THEN
       "Production_HMI".Button_Pop_TODO_To_ENDING.Color := "HMI_COLOR_GREEN";
   END_IF;
END_REGION

REGION Network 27: <+>
END_REGION

REGION Network 28: HMI - Mostra dettagli ordine
END_REGION

REGION Network 29 (SCL): HMI - Mostra dettagli com
   "Production_HMI".Button_ShowDetatails.Show := FALSE;

   IF "Production_HMI".Sel_Index >= 301 THEN
       #indx_Detail := "Production_HMI".Sel_Index - 300;

   ELSIF "Production_HMI".Sel_Index >= 201 THEN
       #indx_Detail := "Production_HMI".Sel_Index - 200;

   ELSIF "Production_HMI".Sel_Index >= 101 THEN
       #indx_Detail := "Production_HMI".Sel_Index - 100;

   ELSIF "Production_HMI".Sel_Index >= 1 THEN
       #indx_Detail := "Production_HMI".Sel_Index;
   END_IF;


   IF #indx_Detail >= 1 AND #indx_Detail <= "PROD_TODO_ITEMS" THEN

       "Production_HMI".Button_ShowDetatails.Show := TRUE;

       IF "Production_HMI".Button_ShowDetatails.Pressed THEN

           "Production_HMI".Button_ShowDetatails.Pressed := FALSE;
           "Production_HMI".Button_ShowDetatails.Show := FALSE;

           IF "Production_HMI".Sel_Index >= 301 THEN
               "Production_HMI".Button_ShowDetatails.Data := "Production".O_OUT[#indx_Detail];

           ELSIF "Production_HMI".Sel_Index >= 201 THEN
               "Production_HMI".Button_ShowDetatails.Data := "Production".O_ENDING[#indx_Detail];

           ELSIF "Production_HMI".Sel_Index >= 101 THEN
               "Production_HMI".Button_ShowDetatails.Data := "Production".O_ACT;

           ELSE
               "Production_HMI".Button_ShowDetatails.Data := "Production".O_TODO[#indx_Detail];
           END_IF;

           #indx_Detail := -1;

       END_IF;

   ELSE
       #indx_Detail := -1;
   END_IF;
END_REGION

REGION Network 30: <+>
END_REGION

REGION Network 31: <+>
END_REGION

REGION Network 32: <+>
END_REGION

REGION Network 33: <+>
END_REGION

REGION Network 36: GESTIONE ACK PER OPERAZIONE DI SETUP MANUALE ESEGUITE
   RUNG wire#powerrail
      #SetUp_Man_Mng(PART_PROD := #PART_PROD, BEAM_PROD := #BEAM_PROD, SET_UP := #SET_UP)
   END_RUNG
   // the same network as SCL:
   #SetUp_Man_Mng(PART_PROD := #PART_PROD, BEAM_PROD := #BEAM_PROD, SET_UP := #SET_UP);   // "Prod_SetUp_Man"
END_REGION

REGION Network 38: >
END_REGION

REGION Network 39: >
END_REGION

REGION Network 40: >
END_REGION

REGION Network 41: >
END_REGION
END_FUNCTION_BLOCK
